// TIA Portal V20 export
VAR_GLOBAL   // PLC tag table "LGR_Const_Task_ComponentID"
END_VAR
VAR_GLOBAL CONSTANT   // user constants
   CompID_GRM : UInt := 4000;
   CompID_GR1 : UInt := 4001;
   CompID_GR2 : UInt := 4002;
   CompID_GCS : UInt := 5000;
   CompID_GR3 : UInt := 4003;
END_VAR
